FUNCTION_BLOCK FB_CART
VAR_INPUT
	stCART: ST_CART;
END_VAR
VAR_OUTPUT
END_VAR

VAR
	inner_counter: INT;
END_VAR

ACTION A_STEP:
IF stCART.position < num_of_carts*2 THEN
	stCART.position:= stCART.position+1;
	stCART.posX:=posArrX[stCART.position];
	stCART.posY:=posArrY[stCART.position];
ELSE
	stCART.position:= 1;
	stCART.posX:=posArrX[stCART.position];
	stCART.posY:=posArrY[stCART.position];
	
END_IF
END_ACTION

END_FUNCTION_BLOCK

(* stored: Version 1.1.0.1, ProductVersion 3.1.4024.12
   POU FB_CART: Id {9fd11ec1-6f9c-4a32-a27f-6e39cedd7563}, SpecialFunc None
   Action A_STEP: Id {14523dd1-b206-4535-943a-bfd0c09ba5ec} *)
